// Monitors the lasers for under voltage events
FUNCTION_BLOCK FB_Laser_Timer
VAR_INPUT
    nVoltageRaw : INT; // The raw signal collected from the ADC
    bAmphosOn : BOOL; // Whether the amphos is turned on
    Timer : TON ; //Timer for reset
    bMasterLatchReset : BOOL; //Master latched error reset
    bCarbideOn : BOOL; // Whether Carbide is ON
    Mode : E_Mode;
END_VAR
VAR_IN_OUT CONSTANT
    stSetpoints : ST_LaserSetpoints; // Setpoints for the laser
END_VAR
VAR_OUTPUT
    {attribute 'pytmc' := '
        pv: VOLTAGE
        io: i
        field: HOPR 10.0
        field: LOPR 0.0
        field: LSV MINOR
        field: LLSV MAJOR
        field: EGU Volts
    '}
    fVoltage : LREAL; // Voltage calculated from the raw ADC input

    {attribute 'pytmc' := '
        pv: SCALED_PWR
        io: i
        field: EGU Watts
    '}
    fPower : LREAL;

    {attribute 'pytmc' := '
        pv: ERROR
        io: i
        field: OSV MAJOR
        field: ZSV NO_ALARM
        field: ZNAM OK
        field: ONAM ERROR
    '}
    bError : BOOL; // Whether an error was detected. Latches until reset
    bBelowNominal : BOOL; //fVoltage is below the nominal setpoint
END_VAR

(* Scale the analog signal to voltage *)
fVoltage := F_Scale(
    fRawData := nVoltageRaw,
    fRawDataLowerOffLimit := GVL_EL3174.fRawLowerLimit,
    fRawDataUpperOffLimit := GVL_EL3174.fRawUpperLimit,
    fScaleDataLowerOffLimit := GVL_EL3174.fScaleLowerLimit,
    fScaleDataUpperOffLimit := GVL_EL3174.fScaleUpperLimit);

fPower := fVoltage; //Value is scaled by user set ASLO and AOFF fields (for display only)

(* Set error if amphos is below nominal voltage *)
IF  (bAmphosOn AND fVoltage < stSetpoints.nMinVoltage) THEN
    Timer(IN:=TRUE, PT:=T#500ms); //500ms SEC Timer
    IF Timer.Q THEN
        bError := TRUE;
        Timer(IN:=FALSE);
    END_IF;
ELSE
    Timer(IN:=FALSE);
END_IF

IF bAmphosOn AND (fVoltage < stSetpoints.nMinNominalVoltage) THEN
    bBelowNominal := TRUE;
END_IF

IF bMasterLatchReset THEN
    bBelowNominal := FALSE;
    bError := FALSE;
END_IF

// Reset latched errors
METHOD Reset
VAR_INPUT
END_VAR
bError := FALSE;
END_METHOD

END_FUNCTION_BLOCK

(* stored: Version 1.1.0.1, ProductVersion 3.1.4024.6
   POU FB_LaserTimer: Id {6b6e0a2c-a634-488b-b528-40d715279b8d}, SpecialFunc None
   Method Reset: Id {f5635c96-77a4-4a28-87e8-262e51f4c847} *)
